// TIA Portal V18 export
DATA_BLOCK "settingsShift"   // DB23
{ S7_Optimized_Access := 'TRUE' }
VERSION : 0.1
// stored: AutoNumber false, DBAccessibleFromOPCUA true, DBAccessibleFromWebserver true, IsOnlyStoredInLoadMemory false, IsRetainMemResEnabled true, IsWriteProtectedInAS false, MemoryReserve 1000, RetainMemoryReserve 1000
   VAR RETAIN
      "1" { ExternalVisible := 'False'; S7_SetPoint := 'True'} : "UDT_settingsShift";
      "2" { ExternalVisible := 'False'; S7_SetPoint := 'True'} : "UDT_settingsShift";
      "3" { ExternalVisible := 'False'; S7_SetPoint := 'True'} : "UDT_settingsShift";
   END_VAR
BEGIN
END_DATA_BLOCK
